FUNCTION_BLOCK ASSEMBLE_AW_FROM_AB (* this Function combines the 2 AB (BYTE) adapters to a AW (WORD) *)
  (* Standard: 61499-2; Description: Copyright (c) 2026 Meisterschulen am Ostbahnhof SPDX-License-Identifier: EPL-2.0 *)
  (* Version 1.0, 2026-05-16, Franz Höpfinger, Meisterschulen am Ostbahnhof, initial API and implementation and/or initial documentation *)
  PACKAGE adapter::assembling;
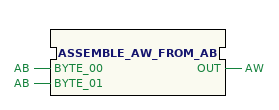
  SOCKETS
    BYTE_00 : adapter::types::unidirectional::AB; (* Byte 0 *)
    BYTE_01 : adapter::types::unidirectional::AB; (* Byte 1 *)
  END_SOCKETS
  PLUGS
    OUT : adapter::types::unidirectional::AW; (* WORD Output *)
  END_PLUGS
END_FUNCTION_BLOCK
